FUNCTION_BLOCK COMPARE_HEXA
VAR_INPUT
	VAR_INTERNAL : UINT;
END_VAR
VAR_OUTPUT
	Error		 : BOOL;
	VAL_3RD_BIT	 : UINT;
	VAL_2ND_BIT	 : UINT;
	VAL_1ST_BIT	 : UINT;
END_VAR
VAR	
END_VAR

IF VAR_INTERNAL >= 16384 AND VAR_INTERNAL < 65356 THEN	
	VAL_3RD_BIT := VAR_INTERNAL/16384;	
	VAL_2ND_BIT := (VAR_INTERNAL - (16384*VAL_3RD_BIT))/64;
	VAL_1ST_BIT := (VAR_INTERNAL - (16384*VAL_3RD_BIT) - (64*VAL_2ND_BIT))*4;
END_IF	
IF VAR_INTERNAL >= 64 AND VAR_INTERNAL < 16384 THEN
	VAL_3RD_BIT := 0;	
	VAL_2ND_BIT := VAR_INTERNAL/64;
	VAL_1ST_BIT := (VAR_INTERNAL - (64*VAL_2ND_BIT))*4;		
END_IF
IF VAR_INTERNAL >= 0 AND VAR_INTERNAL < 64 THEN
	VAL_3RD_BIT := 0;		
	VAL_2ND_BIT := 0;
	VAL_1ST_BIT := VAR_INTERNAL*4;		
END_IF

END_FUNCTION_BLOCK

(* stored: Version 1.1.0.1, ProductVersion 3.1.4024.0
   POU COMPARE_HEXA: Id {9bc626d6-ad7b-4d9f-ae2a-a0a8af42f3db}, SpecialFunc None *)
